{attribute 'Tc2GvlVarNames'}
VAR_GLOBAL PERSISTENT
	(* Axis reference positions *)
	X_REF:LREAL:=0;
	Y_REF:LREAL:=0;

	(* Home position for axis *)
	X_Home:LREAL:=0;
	Y_Home:LREAL:=0;

END_VAR

(* stored: Version 1.1.0.1, ProductVersion 3.1.4024.10
   GVL SETTINGS: Id {503719da-5fb7-41b6-bcc4-466c77c22854} *)
